# EPICS StreamDevice protocol: protocols/hadcon_OWTP_intr.proto
Terminator  = LF;
LockTimeout  = 5000;
ReplyTimeout  = 4000;
ReadTimeout   = 500;
WriteTimeout  = 3000;
ExtraInput    = Ignore;

#
# one wire temperatures
#

OWTP {
# Example of command field(INP, "@<file.proto> OWTP_convert <port>")
	ExtraInput = Ignore;

	out "OWTP";
}

OWTP_err_intr {
	# Example of command field(INP,  "@hadcon_OWTP.proto OWTP_err_intr($(ID)) $(device)")

    in "ERR%*1c OWTP \$1 %39c";
}

OWTP_read_ID_intr {
# Example of command field(INP, "@<file.proto> OWTP_read_ID(28F541F1010000F6) <port>")
	ExtraInput = Ignore;

                     #ID = %\${1};
             #recordName = %\${2};
	Terminator  = CR;

	in "%*{\nRECV|RECV} OWTP \$1 %x";
#	in "RECV OWTP \$1 %x";
}
